(* IEC 61131-3 sources: eCockpitGit/test_project/src/%F%00 Library/%F%Common Functions/%F%Compare, 2 files *)

(* ---- %POU%FU_CompareAny.st ---- *)
//This functions compares two structs, if data in struct are different, then it returns true
//If the two inputs are different sizes, it will compare the amount of bits from the smallest input, to the same amount of bits on the biggest input, and ignore the rest
//FU_CompareStruct(aA:= , aB:= );
// +-----------+----------+----------+-----------------------------------------------------------------------------------------------------------------------+
// |**Version**|**Author**| **Date** |**Changes**                                                                                                            |
// +-----------+----------+----------+-----------------------------------------------------------------------------------------------------------------------+
// | 1         | NSN      | 01-10-18 | Creation                                                                                                              |
// +-----------+----------+----------+-----------------------------------------------------------------------------------------------------------------------+
FUNCTION FU_CompareAny : BOOL
VAR_INPUT
	aA				:ANY;			//Address of first struct
	aB				:ANY;			//Size of first struct in bytes
END_VAR
(*%!%__DELIMITER__%!%*)
IF aA.diSize <= aB.diSize THEN		//Smallest struct is found
	WHILE aA.diSize > 0 DO
		aA.diSize		:=		aA.diSize - 1;
		IF aA.pValue^ <> aB.pValue^ THEN	//Bytes are compared
			FU_CompareAny	:=		TRUE;
		END_IF
		aA.pValue		:=		aA.pValue + 1;
		aB.pValue		:=		aB.pValue + 1;
	END_WHILE
ELSE
	WHILE aB.diSize > 0 DO
		aB.diSize		:=		aB.diSize - 1;
		IF aA.pValue^ <> aB.pValue^ THEN	//Bytes are compared
			FU_CompareAny	:=		TRUE;
		END_IF
		aA.pValue		:=		aA.pValue + 1;
		aB.pValue		:=		aB.pValue + 1;
	END_WHILE
END_IF

(* ---- %POU%FU_CompareStruct.st ---- *)
//This functions compares two structs, if data in struct are different, then it returns true
//FU_CompareStruct(pStructA:= ADR(StructA), uiSizeA:= SIZEOF(StructA), pStructB:= ADR(StructB), uiSizeB:= SIZEOF(StructB));
// +-----------+----------+----------+-----------------------------------------------------------------------------------------------------------------------+
// |**Version**|**Author**| **Date** |**Changes**                                                                                                            |
// +-----------+----------+----------+-----------------------------------------------------------------------------------------------------------------------+
// | 1         | NSN      | 20-12-17 | Creation                                                                                                              |
// +-----------+----------+----------+-----------------------------------------------------------------------------------------------------------------------+
// | 1.1       | NSN      | 13-06-18 | Updated names and types                                                                                               |
// +-----------+----------+----------+-----------------------------------------------------------------------------------------------------------------------+
FUNCTION FU_CompareStruct : bool
VAR_INPUT
	pStructA		:POINTER TO BYTE;		//Address of first struct
	uiSizeA			:UINT;					//Size of first struct in bytes
	pStructB		:POINTER TO BYTE;		//Address of second struct
	uiSizeB			:UINT;					//Size of second struct in bytes
END_VAR
VAR
	FOR1			:WORD;
	LowestSize		:WORD;					//Keeps track of which struct is the smallest, if there is a difference
END_VAR
(*%!%__DELIMITER__%!%*)
IF uiSizeA < uiSizeB THEN		//Smallest struct is found
	LowestSize		:=		uiSizeA;
ELSE
	LowestSize		:=		uiSizeB;
END_IF
WHILE LowestSize > 0 DO
	LowestSize		:=		LowestSize - 1;
	IF pStructA^ <> pStructB^ THEN	//Bytes are compared
		FU_CompareStruct	:=		TRUE;
	END_IF
	pStructA		:=		pStructA + 1;
	pStructB		:=		pStructB + 1;
END_WHILE
